Yaskawa INFORM job: A_NAIHAN_0617_1_PL8.JBI

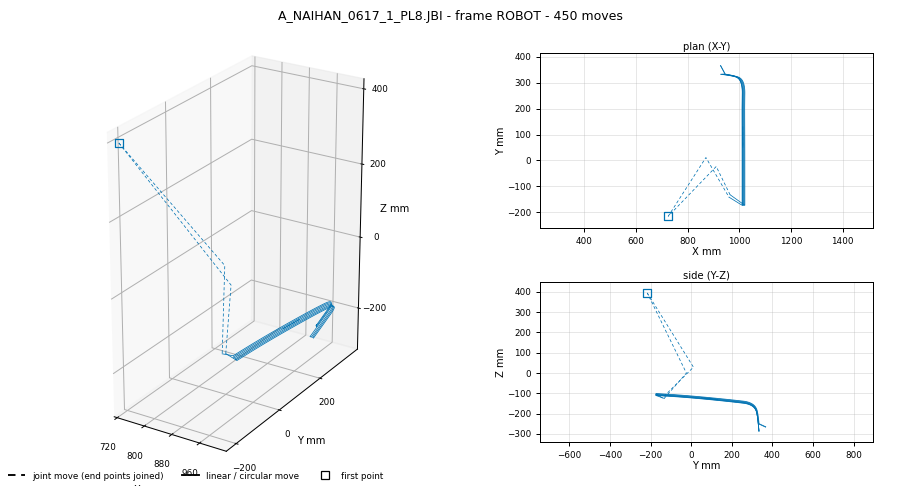
[picture p0: tool path of A_NAIHAN_0617_1_PL8.JBI in frame ROBOT, 450 of 450 moves have a stored position in this frame; points joined in program order, loops and branches not executed]
/JOB
//NAME A_NAIHAN_0617_1
//POS
///NPOS 450,0,0,0,0,0
///TOOL 0
///USER 0
///POSTYPE ROBOT
///RECTAN
///RCONF 0,0,0,0,1,0,0,0,0,0,0,0,0,0,0,0,0,0,0,0,0,0,0,0
C00000=724.889,-216.680,394.500,-180.000,-0.000,-0.000
///USER 0
///POSTYPE ROBOT
///RECTAN
///RCONF 0,0,0,0,1,0,0,0,0,0,0,0,0,0,0,0,0,0,0,0,0,0,0,0
C00001=871.033,10.919,28.927,-91.021,-3.476,-89.989
C00002=960.317,-142.344,-122.679,-91.021,-3.476,-89.989
C00003=1011.126,-173.807,-100.734,-91.021,-3.476,-89.989
C00004=1011.125,-163.825,-101.340,-91.021,-3.476,-89.989
C00005=1011.116,-111.653,-104.509,-90.969,-3.711,-89.998
C00006=1011.118,-93.020,-105.718,-90.950,-3.908,-90.001
C00007=1011.122,-76.836,-106.823,-90.973,-4.109,-90.000
C00008=1011.124,-58.612,-108.132,-91.010,-4.317,-89.996
C00009=1011.125,-38.936,-109.618,-91.108,-4.540,-89.984
C00010=1011.123,-16.317,-111.413,-91.253,-4.759,-89.964
C00011=1011.112,6.932,-113.349,-91.480,-4.971,-89.938
C00012=1011.092,32.226,-115.549,-91.811,-5.168,-89.904
C00013=1011.058,59.070,-117.977,-92.267,-5.359,-89.865
C00014=1011.005,88.104,-120.701,-92.903,-5.531,-89.830
C00015=1010.943,119.307,-123.725,-93.738,-5.698,-89.811
C00016=1010.888,151.031,-126.893,-94.762,-5.867,-89.825
C00017=1010.859,180.841,-129.962,-95.878,-6.031,-89.888
C00018=1010.877,203.531,-132.365,-96.764,-6.194,-90.474
C00019=1011.077,221.566,-134.329,-97.486,-6.326,-90.590
C00020=1011.187,230.412,-135.312,-97.826,-6.451,-90.643
C00021=1011.420,247.118,-137.207,-98.440,-6.622,-90.758
C00022=1011.621,259.754,-138.679,-98.920,-7.725,-90.485
C00023=1011.632,262.262,-139.018,-99.108,-8.924,-89.672
C00024=1011.607,264.768,-139.410,-99.293,-10.096,-88.851
C00025=1011.545,267.269,-139.853,-99.481,-11.298,-88.009
C00026=1011.445,269.766,-140.350,-99.673,-12.511,-87.149
C00027=1011.308,272.257,-140.902,-99.873,-13.722,-86.271
C00028=1011.132,274.742,-141.507,-100.082,-14.960,-85.369
C00029=1010.915,277.219,-142.169,-100.305,-16.218,-84.438
C00030=1010.659,279.689,-142.888,-100.548,-17.483,-83.475
C00031=1010.361,282.148,-143.665,-100.818,-18.811,-82.464
C00032=1010.018,284.597,-144.504,-101.127,-20.211,-81.386
C00033=1009.631,287.030,-145.407,-101.481,-21.679,-80.238
C00034=1009.172,289.568,-146.427,-101.907,-23.208,-78.952
C00035=1008.707,291.848,-147.420,-102.373,-24.814,-77.653
C00036=1008.163,294.223,-148.541,-102.937,-26.542,-76.170
C00037=1007.560,296.570,-149.745,-103.613,-28.449,-74.510
C00038=1006.890,298.869,-151.034,-104.340,-29.973,-72.818
C00039=1006.406,300.387,-151.949,-104.930,-31.287,-71.518
C00040=1005.891,301.885,-152.907,-105.615,-32.677,-70.114
C00041=1005.343,303.357,-153.910,-106.377,-34.082,-68.619
C00042=1004.761,304.804,-154.960,-107.214,-35.486,-67.034
C00043=1004.143,306.220,-156.055,-108.161,-36.921,-65.343
C00044=1003.492,307.602,-157.197,-109.202,-38.372,-63.542
C00045=1002.805,308.949,-158.387,-110.315,-39.727,-61.684
C00046=1002.082,310.261,-159.625,-111.649,-41.378,-59.567
C00047=1001.234,311.656,-161.050,-113.007,-42.578,-57.439
C00048=1000.552,312.697,-162.185,-114.344,-43.933,-55.439
C00049=999.621,314.016,-163.729,-116.012,-45.295,-52.982
C00050=998.687,315.224,-165.258,-117.761,-46.611,-50.477
C00051=997.725,316.363,-166.823,-119.542,-47.783,-47.973
C00052=996.735,317.437,-168.418,-121.388,-48.890,-45.428
C00053=995.722,318.443,-170.040,-123.267,-49.899,-42.881
C00054=994.688,319.382,-171.683,-125.156,-50.806,-40.357
C00055=993.638,320.257,-173.344,-127.088,-51.666,-37.810
C00056=992.574,321.066,-175.019,-129.188,-52.602,-35.078
C00057=990.968,322.171,-177.542,-131.768,-53.377,-31.733
C00058=989.871,322.832,-179.245,-133.513,-53.876,-29.514
C00059=988.772,323.442,-180.948,-135.159,-54.294,-27.432
C00060=987.693,323.993,-182.622,-136.744,-54.682,-25.420
C00061=986.590,324.511,-184.330,-138.472,-55.162,-23.254
C00062=984.951,325.201,-186.860,-140.211,-55.397,-21.070
C00063=983.843,325.624,-188.571,-141.648,-55.749,-19.284
C00064=982.186,326.194,-191.123,-143.265,-56.044,-17.268
C00065=980.003,326.860,-194.483,-144.852,-56.286,-15.287
C00066=977.286,327.590,-198.669,-146.297,-56.550,-13.468
C00067=971.932,328.854,-206.947,-147.090,-56.682,-12.382
C00068=966.688,330.004,-215.111,-147.508,-56.903,-11.777
C00069=961.537,331.076,-223.179,-148.103,-57.125,-10.988
C00070=957.484,331.859,-229.552,-148.860,-57.303,-10.044
C00071=953.493,332.560,-235.849,-149.738,-57.463,-8.963
C00072=949.565,333.173,-242.058,-134.282,-48.007,-28.256
C00073=945.322,333.743,-248.775,-133.027,-46.430,-30.116
C00074=945.165,333.805,-248.991,-133.479,-46.413,-30.686
C00075=944.958,333.955,-249.230,-134.760,-46.419,-32.358
C00076=944.837,334.081,-249.352,-135.802,-46.422,-33.939
C00077=944.742,334.207,-249.441,-136.752,-46.409,-35.644
C00078=944.691,334.289,-249.486,-137.317,-46.388,-36.848
C00079=931.526,358.822,-260.929,-135.450,-44.128,-41.468
C00080=927.152,366.971,-264.731,-134.975,-43.638,-42.153
C00081=928.982,365.318,-266.027,-135.026,-43.691,-42.079
C00082=933.356,357.169,-262.224,-135.507,-44.186,-41.385
C00083=946.521,332.636,-250.782,-137.318,-46.389,-36.846
C00084=946.573,332.553,-250.735,-136.758,-46.414,-35.636
C00085=946.667,332.428,-250.648,-135.814,-46.433,-33.923
C00086=946.787,332.300,-250.526,-134.776,-46.435,-32.336
C00087=946.995,332.152,-250.287,-133.499,-46.434,-30.657
C00088=947.152,332.090,-250.071,-133.049,-46.453,-30.085
C00089=951.383,331.514,-243.366,-134.267,-47.993,-28.276
C00090=955.298,330.902,-237.172,-136.904,-50.492,-24.767
C00091=959.279,330.203,-230.891,-136.971,-50.766,-24.682
C00092=963.321,329.421,-224.533,-136.501,-50.557,-25.308
C00093=968.462,328.349,-216.481,-135.964,-50.158,-26.081
C00094=973.699,327.199,-208.326,-135.696,-49.882,-26.545
C00095=977.957,326.200,-201.731,-135.251,-49.674,-27.196
C00096=979.030,325.933,-200.073,-135.479,-49.973,-26.923
C00097=981.725,325.205,-195.918,-135.092,-50.148,-27.440
C00098=983.890,324.541,-192.580,-134.407,-50.230,-28.313
C00099=985.528,323.974,-190.055,-133.645,-50.246,-29.285
C00100=986.616,323.559,-188.376,-132.921,-50.149,-30.209
C00101=988.232,322.878,-185.878,-131.610,-49.907,-31.885
C00102=989.315,322.369,-184.201,-130.639,-49.725,-33.134
C00103=990.394,321.818,-182.528,-129.535,-49.450,-34.571
C00104=991.468,321.217,-180.857,-128.296,-49.082,-36.173
C00105=992.535,320.563,-179.193,-126.947,-48.616,-37.929
C00106=993.065,320.218,-178.362,-126.262,-48.351,-38.853
C00107=994.117,319.480,-176.711,-124.881,-47.852,-40.674
C00108=995.157,318.685,-175.071,-123.497,-47.333,-42.529
C00109=996.183,317.828,-173.447,-122.066,-46.733,-44.462
C00110=997.191,316.909,-171.842,-120.611,-46.060,-46.454
C00111=998.177,315.925,-170.260,-119.144,-45.318,-48.489
C00112=999.141,314.877,-168.705,-117.682,-44.508,-50.551
C00113=1000.078,313.763,-167.182,-116.238,-43.636,-52.625
C00114=1000.984,312.586,-165.692,-114.824,-42.706,-54.692
C00115=1001.878,311.318,-164.211,-113.432,-41.711,-56.781
C00116=1002.547,310.291,-163.093,-112.384,-40.911,-58.373
C00117=1003.359,308.937,-161.717,-111.135,-39.849,-60.356
C00118=1004.060,307.667,-160.518,-110.055,-38.863,-62.095
C00119=1004.726,306.358,-159.363,-109.064,-37.865,-63.765
C00120=1005.358,305.013,-158.252,-108.147,-36.863,-65.367
C00121=1005.956,303.635,-157.188,-107.298,-35.864,-66.889
C00122=1006.520,302.227,-156.167,-106.538,-34.877,-68.334
C00123=1007.053,300.793,-155.191,-105.843,-33.908,-69.699
C00124=1007.553,299.333,-154.259,-105.214,-32.965,-70.984
C00125=1008.022,297.852,-153.368,-104.664,-32.052,-72.190
C00126=1008.671,295.596,-152.107,-103.923,-30.683,-73.881
C00127=1009.259,293.302,-150.932,-103.280,-29.313,-75.439
C00128=1009.788,290.977,-149.836,-102.723,-27.982,-76.866
C00129=1010.241,288.746,-148.865,-102.264,-26.778,-78.109
C00130=1010.689,286.253,-147.863,-101.826,-25.499,-79.378
C00131=1011.068,283.863,-146.978,-101.464,-24.334,-80.497
C00132=1011.402,281.457,-146.155,-101.147,-23.223,-81.547
C00133=1011.694,279.038,-145.391,-100.867,-22.168,-82.533
C00134=1011.946,276.609,-144.684,-100.614,-21.162,-83.474
C00135=1012.158,274.171,-144.034,-100.382,-20.204,-84.377
C00136=1012.330,271.725,-143.437,-100.165,-19.294,-85.245
C00137=1012.467,269.274,-142.895,-99.957,-18.441,-86.085
C00138=1012.565,266.816,-142.406,-99.760,-17.660,-86.895
C00139=1012.629,264.352,-141.968,-99.569,-16.988,-87.674
C00140=1012.655,261.886,-141.582,-99.387,-16.502,-88.409
C00141=1012.638,258.582,-141.145,-99.174,-16.477,-89.270
C00142=1012.473,246.808,-139.768,-98.759,-16.781,-89.191
C00143=1012.269,230.113,-137.862,-98.090,-15.953,-89.291
C00144=1012.173,221.267,-136.872,-97.724,-15.534,-89.339
C00145=1012.003,202.505,-134.814,-97.004,-15.313,-88.850
C00146=1012.031,180.575,-132.476,-96.047,-14.813,-88.956
C00147=1012.106,150.778,-129.386,-94.882,-13.967,-89.131
C00148=1012.207,119.064,-126.196,-93.817,-13.011,-89.322
C00149=1012.305,87.873,-123.155,-92.956,-12.111,-89.490
C00150=1012.380,58.844,-120.419,-92.302,-11.338,-89.624
C00151=1012.434,32.009,-117.980,-91.836,-10.680,-89.726
C00152=1012.467,6.724,-115.774,-91.497,-10.099,-89.803
C00153=1012.486,-16.516,-113.835,-91.267,-9.615,-89.857
C00154=1012.494,-39.125,-112.036,-91.118,-9.152,-89.894
C00155=1012.498,-58.791,-110.550,-91.019,-8.788,-89.916
C00156=1012.498,-77.004,-109.239,-90.981,-8.477,-89.925
C00157=1012.497,-93.176,-108.133,-90.958,-8.278,-89.928
C00158=1012.497,-111.810,-106.924,-90.977,-8.288,-89.920
C00159=1012.501,-163.972,-103.758,-91.029,-7.712,-89.913
C00160=1012.501,-173.954,-103.153,-91.029,-7.712,-89.913
C00161=1014.014,-174.140,-105.813,-31.342,-6.169,-94.624
C00162=1014.013,-164.159,-106.417,-31.348,-6.135,-94.568
C00163=1014.015,-112.281,-109.562,-31.265,-6.608,-94.935
C00164=1014.017,-90.505,-110.980,-31.253,-6.707,-94.678
C00165=1014.016,-68.918,-112.482,-31.199,-7.017,-94.775
C00166=1014.011,-46.453,-114.145,-31.142,-7.335,-94.876
C00167=1013.998,-23.411,-115.952,-31.075,-7.690,-95.043
C00168=1013.972,0.396,-117.919,-31.002,-8.058,-95.245
C00169=1013.928,25.726,-120.115,-30.912,-8.481,-95.547
C00170=1013.861,52.121,-122.502,-30.810,-8.932,-95.921
C00171=1013.765,80.039,-125.125,-30.690,-9.428,-96.395
C00172=1013.605,120.357,-129.005,-30.456,-10.243,-97.671
C00173=1013.567,130.311,-129.963,-30.383,-10.477,-98.075
C00174=1013.899,50.910,-122.247,-30.789,-9.085,-95.683
C00175=1013.854,60.863,-123.223,-30.709,-9.377,-96.181
C00176=1013.614,115.510,-128.586,-31.175,-10.246,-97.193
C00177=1013.492,141.294,-131.183,-31.903,-10.709,-97.471
C00178=1013.353,171.798,-134.344,-32.900,-11.307,-97.838
C00179=1013.248,202.920,-137.679,-34.238,-11.383,-97.402
C00180=1013.378,220.938,-139.671,-34.793,-11.965,-98.404
C00181=1013.535,237.631,-141.563,-35.328,-12.464,-98.827
C00182=1013.774,258.227,-143.970,-36.132,-12.486,-98.470
C00183=1013.789,260.666,-144.286,-36.310,-13.170,-97.014
C00184=1013.771,263.093,-144.648,-36.487,-13.935,-95.657
C00185=1013.718,265.516,-145.063,-36.656,-14.783,-94.395
C00186=1013.632,267.934,-145.528,-36.819,-15.698,-93.199
C00187=1013.510,270.346,-146.044,-36.986,-16.662,-92.036
C00188=1013.352,272.751,-146.612,-37.162,-17.657,-90.881
C00189=1013.156,275.150,-147.232,-37.355,-18.685,-89.713
C00190=1012.925,277.538,-147.908,-37.565,-19.752,-88.527
C00191=1012.653,279.917,-148.638,-37.798,-20.865,-87.330
C00192=1012.342,282.282,-149.426,-38.065,-22.040,-86.086
C00193=1011.987,284.632,-150.273,-38.376,-23.275,-84.784
C00194=1011.588,286.962,-151.182,-38.744,-24.574,-83.398
C00195=1011.142,289.270,-152.157,-39.190,-25.945,-81.890
C00196=1010.646,291.551,-153.201,-39.732,-27.390,-80.226
C00197=1010.095,293.800,-154.320,-40.395,-28.908,-78.371
C00198=1009.487,296.011,-155.518,-41.217,-30.486,-76.285
C00199=1009.048,297.461,-156.364,-41.874,-31.563,-74.749
C00200=1008.580,298.890,-157.248,-42.631,-32.653,-73.094
C00201=1008.082,300.297,-158.174,-43.478,-33.756,-71.320
C00202=1007.552,301.676,-159.140,-44.447,-34.867,-69.427
C00203=1006.991,303.027,-160.150,-45.520,-35.980,-67.427
C00204=1006.397,304.347,-161.203,-46.700,-37.090,-65.319
C00205=1005.770,305.634,-162.299,-48.003,-38.185,-63.118
C00206=1005.110,306.884,-163.439,-49.400,-39.256,-60.825
C00207=1004.241,308.388,-164.921,-51.285,-40.538,-57.860
C00208=1003.336,309.801,-166.440,-53.291,-41.722,-54.847
C00209=1002.493,311.004,-167.842,-55.157,-42.698,-52.114
C00210=1001.616,312.147,-169.284,-57.091,-43.591,-49.360
C00211=1000.709,313.230,-170.761,-59.067,-44.396,-46.598
C00212=999.776,314.252,-172.271,-61.075,-45.109,-43.854
C00213=998.818,315.212,-173.809,-63.083,-45.731,-41.144
C00214=997.838,316.110,-175.372,-65.087,-46.260,-38.486
C00215=996.840,316.949,-176.955,-67.062,-46.698,-35.897
C00216=995.826,317.729,-178.557,-68.994,-47.054,-33.389
C00217=994.798,318.452,-180.172,-70.866,-47.338,-30.988
C00218=993.369,319.356,-182.408,-73.296,-47.613,-27.880
C00219=992.193,320.022,-184.241,-75.155,-47.743,-25.538
C00220=990.994,320.636,-186.104,-76.899,-47.800,-23.353
C00221=989.796,321.192,-187.962,-78.471,-47.796,-21.379
C00222=988.191,321.859,-190.443,-80.317,-47.727,-19.073
C00223=986.580,322.452,-192.931,-81.869,-47.600,-17.141
C00224=984.970,322.982,-195.416,-83.141,-47.425,-15.558
C00225=983.091,323.538,-198.315,-84.282,-47.192,-14.132
C00226=982.021,323.832,-199.970,-84.780,-47.056,-13.490
C00227=979.883,324.380,-203.271,-85.527,-46.787,-12.542
C00228=975.642,325.379,-209.844,-86.256,-46.530,-11.583
C00229=969.385,326.751,-219.600,-86.681,-46.596,-10.945
C00230=964.277,327.805,-227.614,-87.195,-46.823,-10.283
C00231=960.262,328.567,-233.936,-87.809,-46.746,-9.522
C00232=956.309,329.245,-240.177,-88.531,-46.083,-8.644
C00233=952.422,329.833,-246.330,-89.280,-44.478,-7.744
C00234=933.594,332.352,-276.195,-89.825,-40.728,-7.100
C00235=928.276,333.063,-284.634,-89.826,-40.292,-7.098
C00236=932.405,333.334,-284.766,-83.149,-39.451,-3.524
C00237=937.727,332.564,-276.334,-83.101,-39.929,-3.598
C00238=958.473,329.565,-243.473,-81.333,-46.634,-5.893
C00239=962.772,328.844,-236.682,-80.388,-47.302,-7.020
C00240=967.076,328.034,-229.906,-79.651,-47.309,-7.882
C00241=972.290,326.961,-221.728,-79.076,-47.004,-8.544
C00242=978.595,325.579,-211.901,-78.521,-46.904,-9.191
C00243=982.937,324.559,-205.178,-77.590,-47.273,-10.302
C00244=985.832,323.803,-200.708,-76.309,-47.711,-11.833
C00245=988.186,323.108,-197.080,-74.688,-48.128,-13.777
C00246=990.346,322.377,-193.752,-72.709,-48.320,-16.151
C00247=991.776,321.826,-191.544,-71.084,-48.433,-18.113
C00248=993.198,321.215,-189.346,-69.222,-48.488,-20.373
C00249=994.609,320.535,-187.160,-67.147,-48.447,-22.907
C00250=996.005,319.781,-184.991,-64.871,-48.316,-25.714
C00251=997.376,318.946,-182.852,-62.428,-48.095,-28.760
C00252=998.386,318.265,-181.268,-60.504,-47.867,-31.187
C00253=999.380,317.535,-179.704,-58.529,-47.559,-33.708
C00254=1000.358,316.751,-178.158,-56.522,-47.155,-36.302
C00255=1001.436,315.805,-176.444,-54.247,-46.590,-39.293
C00256=1002.416,314.861,-174.875,-52.143,-45.943,-42.113
C00257=1003.180,314.063,-173.644,-50.477,-45.355,-44.387
C00258=1004.007,313.133,-172.302,-48.652,-44.639,-46.931
C00259=1004.813,312.151,-170.985,-46.864,-43.848,-49.485
C00260=1005.743,310.916,-169.450,-44.803,-42.806,-52.520
C00261=1006.590,309.682,-168.037,-42.954,-41.714,-55.346
C00262=1007.286,308.581,-166.863,-41.473,-40.708,-57.698
C00263=1007.924,307.494,-165.777,-40.139,-39.699,-59.895
C00264=1008.593,306.260,-164.624,-38.785,-38.556,-62.225
C00265=1009.228,304.990,-163.513,-37.543,-37.383,-64.470
C00266=1009.782,303.791,-162.531,-36.504,-36.291,-66.446
C00267=1010.357,302.454,-161.501,-35.478,-35.097,-68.506
C00268=1011.045,300.695,-160.244,-34.330,-33.576,-70.989
C00269=1011.683,298.890,-159.052,-33.361,-32.070,-73.282
C00270=1012.273,297.042,-157.925,-32.563,-30.591,-75.374
C00271=1012.818,295.158,-156.860,-31.916,-29.152,-77.271
C00272=1013.318,293.241,-155.855,-31.401,-27.761,-78.986
C00273=1013.777,291.296,-154.906,-30.996,-26.428,-80.536
C00274=1014.197,289.326,-154.013,-30.678,-25.151,-81.954
C00275=1014.580,287.336,-153.169,-30.432,-23.934,-83.255
C00276=1014.929,285.328,-152.375,-30.245,-22.778,-84.452
C00277=1015.242,283.304,-151.627,-30.101,-21.667,-85.587
C00278=1015.525,281.267,-150.923,-29.992,-20.600,-86.673
C00279=1015.776,279.219,-150.263,-29.912,-19.585,-87.720
C00280=1015.998,277.160,-149.644,-29.851,-18.616,-88.764
C00281=1016.190,275.092,-149.066,-29.803,-17.697,-89.831
C00282=1016.426,271.977,-148.274,-29.782,-16.356,-91.371
C00283=1016.601,268.846,-147.570,-29.838,-15.006,-92.798
C00284=1016.699,266.262,-147.054,-29.918,-13.920,-93.961
C00285=1016.753,263.916,-146.637,-29.998,-13.003,-95.091
C00286=1016.775,261.499,-146.257,-30.077,-12.164,-96.403
C00287=1016.755,258.398,-145.842,-30.170,-11.278,-98.358
C00288=1016.669,251.984,-145.079,-29.920,-11.971,-99.652
C00289=1016.467,235.201,-143.120,-30.101,-11.439,-98.903
C00290=1016.262,213.970,-140.715,-30.322,-10.757,-97.897
C00291=1016.173,202.386,-139.430,-30.410,-10.545,-97.118
C00292=1016.186,195.201,-138.643,-30.442,-10.435,-96.991
C00293=1016.264,167.943,-135.725,-30.495,-10.229,-96.870
C00294=1016.375,138.405,-132.657,-30.623,-9.754,-96.321
C00295=1016.498,107.613,-129.559,-30.757,-9.232,-95.744
C00296=1016.601,78.604,-126.733,-30.871,-8.751,-95.265
C00297=1016.682,50.724,-124.111,-30.969,-8.302,-94.879
C00298=1016.738,24.332,-121.724,-31.053,-7.889,-94.574
C00299=1016.772,-0.206,-119.597,-31.126,-7.509,-94.338
C00300=1016.792,-24.004,-117.630,-31.190,-7.155,-94.164
C00301=1016.801,-46.252,-115.885,-31.247,-6.823,-94.025
C00302=1016.804,-68.716,-114.220,-31.297,-6.513,-93.938
C00303=1016.802,-90.304,-112.717,-31.340,-6.240,-93.906
C00304=1016.800,-112.080,-111.298,-31.360,-6.089,-94.077
C00305=1016.798,-163.958,-108.154,-31.432,-5.635,-93.744
C00306=1016.799,-173.939,-107.550,-31.432,-5.639,-93.750
C00307=1019.319,-173.757,-109.120,-31.722,-3.376,-90.059
C00308=1019.318,-163.775,-109.725,-31.722,-3.376,-90.059
C00309=1019.320,-111.898,-112.869,-31.700,-3.636,-90.066
C00310=1019.323,-90.121,-114.289,-31.679,-3.892,-90.062
C00311=1019.325,-68.534,-115.792,-31.658,-4.146,-90.056
C00312=1019.324,-46.069,-117.458,-31.637,-4.396,-90.037
C00313=1019.317,-23.822,-119.204,-31.616,-4.634,-90.015
C00314=1019.299,-0.024,-121.172,-31.596,-4.867,-89.980
C00315=1019.267,24.514,-123.300,-31.577,-5.085,-89.940
C00316=1019.214,50.907,-125.690,-31.560,-5.295,-89.894
C00317=1019.137,78.787,-128.314,-31.543,-5.495,-89.852
C00318=1019.039,107.798,-131.143,-31.526,-5.684,-89.827
C00319=1018.927,137.765,-134.162,-31.507,-5.873,-89.834
C00320=1018.822,167.327,-137.234,-31.487,-6.066,-89.885
C00321=1018.752,194.584,-140.155,-31.463,-6.261,-89.973
C00322=1018.747,203.291,-141.113,-31.417,-6.531,-90.349
C00323=1018.840,214.653,-142.375,-31.414,-6.444,-90.605
C00324=1019.060,236.382,-144.844,-31.383,-6.658,-90.770
C00325=1019.345,258.586,-147.458,-31.352,-6.876,-90.880
C00326=1019.368,261.687,-147.873,-31.240,-8.353,-89.879
C00327=1019.347,264.103,-148.254,-31.178,-9.499,-89.054
C00328=1019.293,266.449,-148.672,-31.134,-10.626,-88.250
C00329=1019.196,269.034,-149.188,-31.109,-11.875,-87.332
C00330=1019.023,272.165,-149.893,-31.113,-13.414,-86.196
C00331=1018.788,275.280,-150.686,-31.149,-14.996,-85.051
C00332=1018.596,277.348,-151.264,-31.199,-16.071,-84.246
C00333=1018.375,279.407,-151.883,-31.282,-17.145,-83.375
C00334=1018.124,281.456,-152.544,-31.373,-18.280,-82.528
C00335=1017.842,283.493,-153.248,-31.505,-19.434,-81.589
C00336=1017.528,285.516,-153.996,-31.664,-20.640,-80.618
C00337=1017.180,287.525,-154.790,-31.852,-21.904,-79.609
C00338=1016.799,289.515,-155.633,-32.108,-23.208,-78.465
C00339=1016.378,291.484,-156.528,-32.404,-24.607,-77.269
C00340=1015.919,293.429,-157.477,-32.769,-26.070,-75.963
C00341=1015.418,295.346,-158.482,-33.205,-27.629,-74.561
C00342=1014.875,297.230,-159.547,-33.753,-29.239,-72.987
C00343=1014.284,299.079,-160.674,-34.410,-30.920,-71.273
C00344=1013.645,300.884,-161.865,-35.167,-32.686,-69.458
C00345=1012.957,302.642,-163.123,-36.056,-34.498,-67.494
C00346=1012.383,303.980,-164.153,-36.863,-35.925,-65.838
C00347=1011.828,305.178,-165.135,-37.704,-37.220,-64.204
C00348=1011.193,306.448,-166.245,-38.712,-38.629,-62.341
C00349=1010.524,307.681,-167.399,-39.805,-40.034,-60.417
C00350=1009.886,308.770,-168.485,-40.896,-41.288,-58.577
C00351=1009.186,309.879,-169.667,-42.090,-42.608,-56.632
C00352=1008.735,310.548,-170.421,-42.979,-43.311,-55.239
C00353=1007.776,311.872,-172.011,-44.729,-44.851,-52.568
C00354=1006.977,312.881,-173.322,-46.245,-45.987,-50.333
C00355=1006.008,314.002,-174.897,-48.072,-47.267,-47.715
C00356=1005.017,315.049,-176.496,-49.965,-48.438,-45.080
C00357=1004.156,315.881,-177.873,-51.608,-49.350,-42.842
C00358=1003.279,316.666,-179.268,-53.299,-50.164,-40.581
C00359=1002.146,317.594,-181.062,-55.415,-51.144,-37.802
C00360=1001.153,318.334,-182.624,-57.269,-51.858,-35.405
C00361=999.804,319.243,-184.738,-59.681,-52.731,-32.334
C00362=998.427,320.069,-186.885,-62.036,-53.468,-29.379
C00363=997.027,320.815,-189.058,-64.262,-54.107,-26.616
C00364=995.614,321.485,-191.247,-66.347,-54.601,-24.054
C00365=994.149,322.104,-193.509,-68.265,-55.040,-21.713
C00366=992.223,322.820,-196.479,-70.424,-55.478,-19.098
C00367=990.783,323.297,-198.698,-71.760,-55.727,-17.488
C00368=988.428,323.991,-202.326,-73.432,-56.049,-15.480
C00369=985.532,324.746,-206.795,-74.751,-56.332,-13.903
C00370=981.189,325.767,-213.518,-75.685,-56.640,-12.788
C00371=974.883,327.149,-223.345,-76.320,-56.877,-12.031
C00372=969.668,328.221,-231.522,-77.053,-57.068,-11.159
C00373=965.365,329.031,-238.298,-77.924,-57.231,-10.123
C00374=961.066,329.753,-245.088,-78.931,-57.390,-8.927
C00375=941.249,332.666,-276.466,-82.914,-40.105,-3.817
C00376=935.927,333.448,-284.896,-82.966,-39.602,-3.736
C00377=938.284,333.676,-286.363,-82.965,-39.613,-3.738
C00378=943.607,332.881,-277.934,-82.913,-40.113,-3.819
C00379=963.423,329.924,-246.563,-81.306,-46.802,-5.930
C00380=967.722,329.201,-239.775,-80.373,-47.379,-7.039
C00381=972.023,328.393,-233.002,-79.639,-47.370,-7.898
C00382=977.234,327.322,-224.830,-79.057,-47.096,-8.570
C00383=983.537,325.941,-215.008,-78.489,-47.048,-9.234
C00384=987.879,324.920,-208.286,-77.547,-47.454,-10.361
C00385=990.776,324.165,-203.816,-76.257,-47.905,-11.903
C00386=993.133,323.471,-200.185,-74.623,-48.338,-13.864
C00387=994.574,323.005,-197.962,-73.349,-48.498,-15.394
C00388=996.503,322.280,-194.990,-71.284,-48.602,-17.879
C00389=997.971,321.661,-192.722,-69.400,-48.661,-20.166
C00390=999.387,320.989,-190.528,-67.352,-48.612,-22.665
C00391=1000.792,320.240,-188.347,-65.102,-48.471,-25.436
C00392=1002.174,319.412,-186.192,-62.675,-48.245,-28.457
C00393=1003.533,318.494,-184.063,-60.106,-47.931,-31.698
C00394=1004.532,317.749,-182.492,-58.124,-47.596,-34.234
C00395=1005.671,316.817,-180.689,-55.785,-47.088,-37.269
C00396=1006.553,316.021,-179.286,-53.933,-46.593,-39.714
C00397=1007.412,315.185,-177.910,-52.094,-46.003,-42.180
C00398=1008.415,314.127,-176.294,-49.942,-45.206,-45.127
C00399=1009.388,312.998,-174.711,-47.813,-44.313,-48.122
C00400=1010.194,311.979,-173.389,-46.052,-43.469,-50.668
C00401=1011.158,310.642,-171.792,-43.952,-42.315,-53.807
C00402=1011.607,309.965,-171.043,-42.980,-41.707,-55.306
C00403=1012.312,308.842,-169.854,-41.504,-40.675,-57.650
C00404=1012.953,307.743,-168.762,-40.188,-39.649,-59.818
C00405=1013.624,306.496,-167.604,-38.851,-38.488,-62.118
C00406=1014.263,305.212,-166.490,-37.627,-37.298,-64.332
C00407=1014.820,304.000,-165.504,-36.603,-36.191,-66.279
C00408=1015.394,302.649,-164.472,-35.592,-34.981,-68.309
C00409=1016.084,300.875,-163.213,-34.457,-33.445,-70.759
C00410=1016.723,299.052,-162.021,-33.496,-31.927,-73.027
C00411=1017.312,297.188,-160.894,-32.700,-30.443,-75.104
C00412=1017.856,295.288,-159.831,-32.049,-29.003,-76.999
C00413=1018.355,293.356,-158.828,-31.524,-27.616,-78.720
C00414=1018.812,291.398,-157.882,-31.109,-26.291,-80.281
C00415=1019.229,289.417,-156.991,-30.780,-25.021,-81.714
C00416=1019.609,287.415,-156.152,-30.524,-23.812,-83.029
C00417=1019.954,285.396,-155.361,-30.327,-22.664,-84.240
C00418=1020.264,283.363,-154.617,-30.175,-21.558,-85.385
C00419=1020.543,281.316,-153.918,-30.061,-20.495,-86.479
C00420=1020.791,279.259,-153.262,-29.976,-19.482,-87.530
C00421=1021.009,277.192,-152.648,-29.912,-18.512,-88.574
C00422=1021.198,275.117,-152.075,-29.860,-17.594,-89.642
C00423=1021.428,271.992,-151.289,-29.831,-16.262,-91.200
C00424=1021.596,268.852,-150.592,-29.883,-14.907,-92.620
C00425=1021.688,266.259,-150.084,-29.969,-13.800,-93.748
C00426=1021.736,263.907,-149.673,-30.057,-12.857,-94.832
C00427=1021.753,261.484,-149.300,-30.142,-11.985,-96.090
C00428=1021.724,258.378,-148.892,-30.245,-11.056,-97.969
C00429=1021.437,236.185,-146.285,-30.142,-11.325,-98.693
C00430=1021.216,214.466,-143.818,-30.336,-10.715,-97.818
C00431=1021.120,202.400,-142.476,-30.422,-10.508,-97.054
C00432=1021.129,194.437,-141.601,-30.458,-10.383,-96.907
C00433=1021.199,167.186,-138.681,-30.519,-10.146,-96.732
C00434=1021.303,137.630,-135.610,-30.647,-9.671,-96.187
C00435=1021.414,107.661,-132.592,-30.772,-9.180,-95.654
C00436=1021.512,78.654,-129.764,-30.881,-8.713,-95.200
C00437=1021.588,50.777,-127.141,-30.976,-8.275,-94.833
C00438=1021.640,24.388,-124.752,-31.058,-7.869,-94.541
C00439=1021.672,-0.146,-122.626,-31.129,-7.497,-94.318
C00440=1021.689,-23.940,-120.659,-31.192,-7.144,-94.146
C00441=1021.696,-46.183,-118.915,-31.248,-6.820,-94.019
C00442=1021.697,-68.642,-117.250,-31.297,-6.515,-93.941
C00443=1021.695,-90.223,-115.748,-31.337,-6.254,-93.929
C00444=1021.691,-111.993,-114.330,-31.359,-6.094,-94.086
C00445=1021.687,-163.864,-111.188,-31.428,-5.660,-93.786
C00446=1021.687,-173.845,-110.584,-31.430,-5.651,-93.771
C00447=964.557,-133.081,-124.802,-31.430,-5.651,-93.771
C00448=910.956,-23.753,-0.173,-31.430,-5.651,-93.771
///USER 0
///POSTYPE ROBOT
///RECTAN
///RCONF 0,0,0,1,1,0,0,0,0,0,0,0,0,0,0,0,0,0,0,0,0,0,0,0
C00449=724.889,-216.680,394.500,-180.000,-0.000,-0.000
//INST
///DATE 2021/06/17 15:04
///ATTR SC,RW,RJ
////FRAME ROBOT1
///GROUP1 RB1
NOP
MOVJ C00000 VJ=100.00 PL=0
'Path Start: Op_ID_1
MOVJ C00001 VJ=25.00 PL=0
MOVJ C00002 VJ=25.00 PL=0
MOVL C00003 V=100.0 PL=0
MOVL C00004 V=800.0 PL=8
SPYON
MOVL C00005 V=800.0 PL=8
MOVL C00006 V=800.0 PL=8
MOVL C00007 V=800.0 PL=8
MOVL C00008 V=800.0 PL=8
MOVL C00009 V=800.0 PL=8
MOVL C00010 V=800.0 PL=8
MOVL C00011 V=800.0 PL=8
MOVL C00012 V=800.0 PL=8
MOVL C00013 V=800.0 PL=8
MOVL C00014 V=800.0 PL=8
MOVL C00015 V=800.0 PL=8
MOVL C00016 V=800.0 PL=8
MOVL C00017 V=800.0 PL=8
MOVL C00018 V=800.0 PL=8
MOVL C00019 V=800.0 PL=8
MOVL C00020 V=800.0 PL=8
MOVL C00021 V=800.0 PL=8
MOVL C00022 V=800.0 PL=8
MOVL C00023 V=800.0 PL=8
MOVL C00024 V=800.0 PL=8
MOVL C00025 V=800.0 PL=8
MOVL C00026 V=800.0 PL=8
MOVL C00027 V=800.0 PL=8
MOVL C00028 V=800.0 PL=8
MOVL C00029 V=800.0 PL=8
MOVL C00030 V=800.0 PL=8
MOVL C00031 V=800.0 PL=8
MOVL C00032 V=800.0 PL=8
MOVL C00033 V=800.0 PL=8
MOVL C00034 V=800.0 PL=8
MOVL C00035 V=800.0 PL=8
MOVL C00036 V=800.0 PL=8
MOVL C00037 V=800.0 PL=8
MOVL C00038 V=800.0 PL=8
MOVL C00039 V=800.0 PL=8
MOVL C00040 V=800.0 PL=8
MOVL C00041 V=800.0 PL=8
MOVL C00042 V=800.0 PL=8
MOVL C00043 V=800.0 PL=8
MOVL C00044 V=800.0 PL=8
MOVL C00045 V=800.0 PL=8
MOVL C00046 V=800.0 PL=8
MOVL C00047 V=800.0 PL=8
MOVL C00048 V=800.0 PL=8
MOVL C00049 V=800.0 PL=8
MOVL C00050 V=800.0 PL=8
MOVL C00051 V=800.0 PL=8
MOVL C00052 V=800.0 PL=8
MOVL C00053 V=800.0 PL=8
MOVL C00054 V=800.0 PL=8
MOVL C00055 V=800.0 PL=8
MOVL C00056 V=800.0 PL=8
MOVL C00057 V=800.0 PL=8
MOVL C00058 V=800.0 PL=8
MOVL C00059 V=800.0 PL=8
MOVL C00060 V=800.0 PL=8
MOVL C00061 V=800.0 PL=8
MOVL C00062 V=800.0 PL=8
MOVL C00063 V=800.0 PL=8
MOVL C00064 V=800.0 PL=8
MOVL C00065 V=800.0 PL=8
MOVL C00066 V=800.0 PL=8
MOVL C00067 V=800.0 PL=8
MOVL C00068 V=800.0 PL=8
MOVL C00069 V=800.0 PL=8
MOVL C00070 V=800.0 PL=8
MOVL C00071 V=800.0 PL=8
MOVL C00072 V=800.0 PL=8
MOVL C00073 V=800.0 PL=8
MOVL C00074 V=800.0 PL=8
MOVL C00075 V=800.0 PL=8
MOVL C00076 V=800.0 PL=8
MOVL C00077 V=800.0 PL=8
MOVL C00078 V=800.0 PL=8
MOVL C00079 V=800.0 PL=8
SPYOF
MOVL C00080 V=800.0 PL=0
MOVJ C00081 VJ=25.00 PL=0
MOVL C00082 V=800.0 PL=8
SPYON
MOVL C00083 V=800.0 PL=8
MOVL C00084 V=800.0 PL=8
MOVL C00085 V=800.0 PL=8
MOVL C00086 V=800.0 PL=8
MOVL C00087 V=800.0 PL=8
MOVL C00088 V=800.0 PL=8
MOVL C00089 V=800.0 PL=8
MOVL C00090 V=800.0 PL=8
MOVL C00091 V=800.0 PL=8
MOVL C00092 V=800.0 PL=8
MOVL C00093 V=800.0 PL=8
MOVL C00094 V=800.0 PL=8
MOVL C00095 V=800.0 PL=8
MOVL C00096 V=800.0 PL=8
MOVL C00097 V=800.0 PL=8
MOVL C00098 V=800.0 PL=8
MOVL C00099 V=800.0 PL=8
MOVL C00100 V=800.0 PL=8
MOVL C00101 V=800.0 PL=8
MOVL C00102 V=800.0 PL=8
MOVL C00103 V=800.0 PL=8
MOVL C00104 V=800.0 PL=8
MOVL C00105 V=800.0 PL=8
MOVL C00106 V=800.0 PL=8
MOVL C00107 V=800.0 PL=8
MOVL C00108 V=800.0 PL=8
MOVL C00109 V=800.0 PL=8
MOVL C00110 V=800.0 PL=8
MOVL C00111 V=800.0 PL=8
MOVL C00112 V=800.0 PL=8
MOVL C00113 V=800.0 PL=8
MOVL C00114 V=800.0 PL=8
MOVL C00115 V=800.0 PL=8
MOVL C00116 V=800.0 PL=8
MOVL C00117 V=800.0 PL=8
MOVL C00118 V=800.0 PL=8
MOVL C00119 V=800.0 PL=8
MOVL C00120 V=800.0 PL=8
MOVL C00121 V=800.0 PL=8
MOVL C00122 V=800.0 PL=8
MOVL C00123 V=800.0 PL=8
MOVL C00124 V=800.0 PL=8
MOVL C00125 V=800.0 PL=8
MOVL C00126 V=800.0 PL=8
MOVL C00127 V=800.0 PL=8
MOVL C00128 V=800.0 PL=8
MOVL C00129 V=800.0 PL=8
MOVL C00130 V=800.0 PL=8
MOVL C00131 V=800.0 PL=8
MOVL C00132 V=800.0 PL=8
MOVL C00133 V=800.0 PL=8
MOVL C00134 V=800.0 PL=8
MOVL C00135 V=800.0 PL=8
MOVL C00136 V=800.0 PL=8
MOVL C00137 V=800.0 PL=8
MOVL C00138 V=800.0 PL=8
MOVL C00139 V=800.0 PL=8
MOVL C00140 V=800.0 PL=8
MOVL C00141 V=800.0 PL=8
MOVL C00142 V=800.0 PL=8
MOVL C00143 V=800.0 PL=8
MOVL C00144 V=800.0 PL=8
MOVL C00145 V=800.0 PL=8
MOVL C00146 V=800.0 PL=8
MOVL C00147 V=800.0 PL=8
MOVL C00148 V=800.0 PL=8
MOVL C00149 V=800.0 PL=8
MOVL C00150 V=800.0 PL=8
MOVL C00151 V=800.0 PL=8
MOVL C00152 V=800.0 PL=8
MOVL C00153 V=800.0 PL=8
MOVL C00154 V=800.0 PL=8
MOVL C00155 V=800.0 PL=8
MOVL C00156 V=800.0 PL=8
MOVL C00157 V=800.0 PL=8
MOVL C00158 V=800.0 PL=8
MOVL C00159 V=800.0 PL=8
SPYOF
MOVL C00160 V=800.0 PL=0
MOVJ C00161 VJ=25.00 PL=0
MOVL C00162 V=800.0 PL=8
SPYON
MOVL C00163 V=800.0 PL=8
MOVL C00164 V=800.0 PL=8
MOVL C00165 V=800.0 PL=8
MOVL C00166 V=800.0 PL=8
MOVL C00167 V=800.0 PL=8
MOVL C00168 V=800.0 PL=8
MOVL C00169 V=800.0 PL=8
MOVL C00170 V=800.0 PL=8
MOVL C00171 V=800.0 PL=8
MOVL C00172 V=800.0 PL=8
SPYOF
MOVL C00173 V=800.0 PL=0
MOVJ C00174 VJ=25.00 PL=0
MOVL C00175 V=800.0 PL=8
SPYON
MOVL C00176 V=800.0 PL=8
MOVL C00177 V=800.0 PL=8
MOVL C00178 V=800.0 PL=8
MOVL C00179 V=800.0 PL=8
MOVL C00180 V=800.0 PL=8
MOVL C00181 V=800.0 PL=8
MOVL C00182 V=800.0 PL=8
MOVL C00183 V=800.0 PL=8
MOVL C00184 V=800.0 PL=8
MOVL C00185 V=800.0 PL=8
MOVL C00186 V=800.0 PL=8
MOVL C00187 V=800.0 PL=8
MOVL C00188 V=800.0 PL=8
MOVL C00189 V=800.0 PL=8
MOVL C00190 V=800.0 PL=8
MOVL C00191 V=800.0 PL=8
MOVL C00192 V=800.0 PL=8
MOVL C00193 V=800.0 PL=8
MOVL C00194 V=800.0 PL=8
MOVL C00195 V=800.0 PL=8
MOVL C00196 V=800.0 PL=8
MOVL C00197 V=800.0 PL=8
MOVL C00198 V=800.0 PL=8
MOVL C00199 V=800.0 PL=8
MOVL C00200 V=800.0 PL=8
MOVL C00201 V=800.0 PL=8
MOVL C00202 V=800.0 PL=8
MOVL C00203 V=800.0 PL=8
MOVL C00204 V=800.0 PL=8
MOVL C00205 V=800.0 PL=8
MOVL C00206 V=800.0 PL=8
MOVL C00207 V=800.0 PL=8
MOVL C00208 V=800.0 PL=8
MOVL C00209 V=800.0 PL=8
MOVL C00210 V=800.0 PL=8
MOVL C00211 V=800.0 PL=8
MOVL C00212 V=800.0 PL=8
MOVL C00213 V=800.0 PL=8
MOVL C00214 V=800.0 PL=8
MOVL C00215 V=800.0 PL=8
MOVL C00216 V=800.0 PL=8
MOVL C00217 V=800.0 PL=8
MOVL C00218 V=800.0 PL=8
MOVL C00219 V=800.0 PL=8
MOVL C00220 V=800.0 PL=8
MOVL C00221 V=800.0 PL=8
MOVL C00222 V=800.0 PL=8
MOVL C00223 V=800.0 PL=8
MOVL C00224 V=800.0 PL=8
MOVL C00225 V=800.0 PL=8
MOVL C00226 V=800.0 PL=8
MOVL C00227 V=800.0 PL=8
MOVL C00228 V=800.0 PL=8
MOVL C00229 V=800.0 PL=8
MOVL C00230 V=800.0 PL=8
MOVL C00231 V=800.0 PL=8
MOVL C00232 V=800.0 PL=8
MOVL C00233 V=800.0 PL=8
MOVL C00234 V=800.0 PL=8
SPYOF
MOVL C00235 V=800.0 PL=0
MOVJ C00236 VJ=25.00 PL=0
MOVL C00237 V=800.0 PL=8
SPYON
MOVL C00238 V=800.0 PL=8
MOVL C00239 V=800.0 PL=8
MOVL C00240 V=800.0 PL=8
MOVL C00241 V=800.0 PL=8
MOVL C00242 V=800.0 PL=8
MOVL C00243 V=800.0 PL=8
MOVL C00244 V=800.0 PL=8
MOVL C00245 V=800.0 PL=8
MOVL C00246 V=800.0 PL=8
MOVL C00247 V=800.0 PL=8
MOVL C00248 V=800.0 PL=8
MOVL C00249 V=800.0 PL=8
MOVL C00250 V=800.0 PL=8
MOVL C00251 V=800.0 PL=8
MOVL C00252 V=800.0 PL=8
MOVL C00253 V=800.0 PL=8
MOVL C00254 V=800.0 PL=8
MOVL C00255 V=800.0 PL=8
MOVL C00256 V=800.0 PL=8
MOVL C00257 V=800.0 PL=8
MOVL C00258 V=800.0 PL=8
MOVL C00259 V=800.0 PL=8
MOVL C00260 V=800.0 PL=8
MOVL C00261 V=800.0 PL=8
MOVL C00262 V=800.0 PL=8
MOVL C00263 V=800.0 PL=8
MOVL C00264 V=800.0 PL=8
MOVL C00265 V=800.0 PL=8
MOVL C00266 V=800.0 PL=8
MOVL C00267 V=800.0 PL=8
MOVL C00268 V=800.0 PL=8
MOVL C00269 V=800.0 PL=8
MOVL C00270 V=800.0 PL=8
MOVL C00271 V=800.0 PL=8
MOVL C00272 V=800.0 PL=8
MOVL C00273 V=800.0 PL=8
MOVL C00274 V=800.0 PL=8
MOVL C00275 V=800.0 PL=8
MOVL C00276 V=800.0 PL=8
MOVL C00277 V=800.0 PL=8
MOVL C00278 V=800.0 PL=8
MOVL C00279 V=800.0 PL=8
MOVL C00280 V=800.0 PL=8
MOVL C00281 V=800.0 PL=8
MOVL C00282 V=800.0 PL=8
MOVL C00283 V=800.0 PL=8
MOVL C00284 V=800.0 PL=8
MOVL C00285 V=800.0 PL=8
MOVL C00286 V=800.0 PL=8
MOVL C00287 V=800.0 PL=8
MOVL C00288 V=800.0 PL=8
MOVL C00289 V=800.0 PL=8
MOVL C00290 V=800.0 PL=8
MOVL C00291 V=800.0 PL=8
MOVL C00292 V=800.0 PL=8
MOVL C00293 V=800.0 PL=8
MOVL C00294 V=800.0 PL=8
MOVL C00295 V=800.0 PL=8
MOVL C00296 V=800.0 PL=8
MOVL C00297 V=800.0 PL=8
MOVL C00298 V=800.0 PL=8
MOVL C00299 V=800.0 PL=8
MOVL C00300 V=800.0 PL=8
MOVL C00301 V=800.0 PL=8
MOVL C00302 V=800.0 PL=8
MOVL C00303 V=800.0 PL=8
MOVL C00304 V=800.0 PL=8
MOVL C00305 V=800.0 PL=8
SPYOF
MOVL C00306 V=800.0 PL=0
MOVJ C00307 VJ=25.00 PL=0
MOVL C00308 V=800.0 PL=8
SPYON
MOVL C00309 V=800.0 PL=8
MOVL C00310 V=800.0 PL=8
MOVL C00311 V=800.0 PL=8
MOVL C00312 V=800.0 PL=8
MOVL C00313 V=800.0 PL=8
MOVL C00314 V=800.0 PL=8
MOVL C00315 V=800.0 PL=8
MOVL C00316 V=800.0 PL=8
MOVL C00317 V=800.0 PL=8
MOVL C00318 V=800.0 PL=8
MOVL C00319 V=800.0 PL=8
MOVL C00320 V=800.0 PL=8
MOVL C00321 V=800.0 PL=8
MOVL C00322 V=800.0 PL=8
MOVL C00323 V=800.0 PL=8
MOVL C00324 V=800.0 PL=8
MOVL C00325 V=800.0 PL=8
MOVL C00326 V=800.0 PL=8
MOVL C00327 V=800.0 PL=8
MOVL C00328 V=800.0 PL=8
MOVL C00329 V=800.0 PL=8
MOVL C00330 V=800.0 PL=8
MOVL C00331 V=800.0 PL=8
MOVL C00332 V=800.0 PL=8
MOVL C00333 V=800.0 PL=8
MOVL C00334 V=800.0 PL=8
MOVL C00335 V=800.0 PL=8
MOVL C00336 V=800.0 PL=8
MOVL C00337 V=800.0 PL=8
MOVL C00338 V=800.0 PL=8
MOVL C00339 V=800.0 PL=8
MOVL C00340 V=800.0 PL=8
MOVL C00341 V=800.0 PL=8
MOVL C00342 V=800.0 PL=8
MOVL C00343 V=800.0 PL=8
MOVL C00344 V=800.0 PL=8
MOVL C00345 V=800.0 PL=8
MOVL C00346 V=800.0 PL=8
MOVL C00347 V=800.0 PL=8
MOVL C00348 V=800.0 PL=8
MOVL C00349 V=800.0 PL=8
MOVL C00350 V=800.0 PL=8
MOVL C00351 V=800.0 PL=8
MOVL C00352 V=800.0 PL=8
MOVL C00353 V=800.0 PL=8
MOVL C00354 V=800.0 PL=8
MOVL C00355 V=800.0 PL=8
MOVL C00356 V=800.0 PL=8
MOVL C00357 V=800.0 PL=8
MOVL C00358 V=800.0 PL=8
MOVL C00359 V=800.0 PL=8
MOVL C00360 V=800.0 PL=8
MOVL C00361 V=800.0 PL=8
MOVL C00362 V=800.0 PL=8
MOVL C00363 V=800.0 PL=8
MOVL C00364 V=800.0 PL=8
MOVL C00365 V=800.0 PL=8
MOVL C00366 V=800.0 PL=8
MOVL C00367 V=800.0 PL=8
MOVL C00368 V=800.0 PL=8
MOVL C00369 V=800.0 PL=8
MOVL C00370 V=800.0 PL=8
MOVL C00371 V=800.0 PL=8
MOVL C00372 V=800.0 PL=8
MOVL C00373 V=800.0 PL=8
MOVL C00374 V=800.0 PL=8
MOVL C00375 V=800.0 PL=8
SPYOF
MOVL C00376 V=800.0 PL=0
MOVJ C00377 VJ=25.00 PL=0
MOVL C00378 V=800.0 PL=8
SPYON
MOVL C00379 V=800.0 PL=8
MOVL C00380 V=800.0 PL=8
MOVL C00381 V=800.0 PL=8
MOVL C00382 V=800.0 PL=8
MOVL C00383 V=800.0 PL=8
MOVL C00384 V=800.0 PL=8
MOVL C00385 V=800.0 PL=8
MOVL C00386 V=800.0 PL=8
MOVL C00387 V=800.0 PL=8
MOVL C00388 V=800.0 PL=8
MOVL C00389 V=800.0 PL=8
MOVL C00390 V=800.0 PL=8
MOVL C00391 V=800.0 PL=8
MOVL C00392 V=800.0 PL=8
MOVL C00393 V=800.0 PL=8
MOVL C00394 V=800.0 PL=8
MOVL C00395 V=800.0 PL=8
MOVL C00396 V=800.0 PL=8
MOVL C00397 V=800.0 PL=8
MOVL C00398 V=800.0 PL=8
MOVL C00399 V=800.0 PL=8
MOVL C00400 V=800.0 PL=8
MOVL C00401 V=800.0 PL=8
MOVL C00402 V=800.0 PL=8
MOVL C00403 V=800.0 PL=8
MOVL C00404 V=800.0 PL=8
MOVL C00405 V=800.0 PL=8
MOVL C00406 V=800.0 PL=8
MOVL C00407 V=800.0 PL=8
MOVL C00408 V=800.0 PL=8
MOVL C00409 V=800.0 PL=8
MOVL C00410 V=800.0 PL=8
MOVL C00411 V=800.0 PL=8
MOVL C00412 V=800.0 PL=8
MOVL C00413 V=800.0 PL=8
MOVL C00414 V=800.0 PL=8
MOVL C00415 V=800.0 PL=8
MOVL C00416 V=800.0 PL=8
MOVL C00417 V=800.0 PL=8
MOVL C00418 V=800.0 PL=8
MOVL C00419 V=800.0 PL=8
MOVL C00420 V=800.0 PL=8
MOVL C00421 V=800.0 PL=8
MOVL C00422 V=800.0 PL=8
MOVL C00423 V=800.0 PL=8
MOVL C00424 V=800.0 PL=8
MOVL C00425 V=800.0 PL=8
MOVL C00426 V=800.0 PL=8
MOVL C00427 V=800.0 PL=8
MOVL C00428 V=800.0 PL=8
MOVL C00429 V=800.0 PL=8
MOVL C00430 V=800.0 PL=8
MOVL C00431 V=800.0 PL=8
MOVL C00432 V=800.0 PL=8
MOVL C00433 V=800.0 PL=8
MOVL C00434 V=800.0 PL=8
MOVL C00435 V=800.0 PL=8
MOVL C00436 V=800.0 PL=8
MOVL C00437 V=800.0 PL=8
MOVL C00438 V=800.0 PL=8
MOVL C00439 V=800.0 PL=8
MOVL C00440 V=800.0 PL=8
MOVL C00441 V=800.0 PL=8
MOVL C00442 V=800.0 PL=8
MOVL C00443 V=800.0 PL=8
MOVL C00444 V=800.0 PL=8
MOVL C00445 V=800.0 PL=8
SPYOF
MOVL C00446 V=800.0 PL=0
MOVL C00447 V=100.0 PL=0
MOVJ C00448 VJ=25.00 PL=0
'Path End
MOVJ C00449 VJ=100.00 PL=0
END
